TYPE ST_PIZZA :
STRUCT
	bExist : BOOL;
	dtTimeEnteredOven : DT;
	dtTimeExitedOven : DT;
	tTimeInOven : TIME;
	eType : E_PIZZA_TYPES; // 0 = Cheese, 1 = Pep, 2 = sausage
	
END_STRUCT
END_TYPE

(* stored: Version 1.1.0.1, ProductVersion 3.1.0.26
   DUT ST_PIZZA: Id {c3bd4980-10fb-41d4-a440-58646530c8f9} *)
